ABB RobotStudio station: SmartComponentSolution_20201017-192109.rsstn

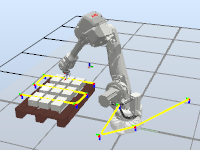
Station SmartComponentSolution (saved by RobotStudio 20.2.9116.0)
Controller IRB_4600_60kg_2.05m, task T_ROB1: task frame (RAPID world) sits at (1429.89, 1152.71, -186.83) mm in the station
Controller IRB_4600_60kg_2.05m
  mechanical unit ROB_1: IRB4600_60_205_C_01, 6 joints, base frame (0, 0, 0) mm
Layout (positions relative to the parent item):
  - IRB4600_60_205_C_01 [mechanism, from Robots\IRB4600_60_205_C_G_01.rslib] at (1429.89, 1152.71, -186.83) mm; joint values [-1.8714, 0.3114, 0.6168, 0, 0.6426, 1.2702] (rad or m)
  - SC_VacuumGripper [smart component] at (3099.75, 399.59, 421.5) mm, rotated rx -180 ry 0 rz 0 deg
      signals: DI diAttach, DO doAttached
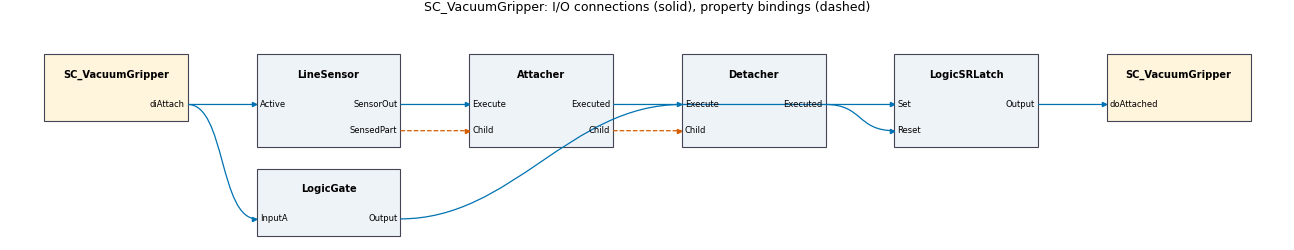
      connections:
        SC_VacuumGripper.diAttach -> LineSensor.Active
        LineSensor.SensorOut -> Attacher.Execute
        SC_VacuumGripper.diAttach -> LogicGate.InputA
        LogicGate.Output -> Detacher.Execute
        Attacher.Executed -> LogicSRLatch.Set
        Detacher.Executed -> LogicSRLatch.Reset
        LogicSRLatch.Output -> SC_VacuumGripper.doAttached
        LineSensor.SensedPart => Attacher.Child
        Attacher.Child => Detacher.Child
    - small_suction_gripper_2 [mechanism] at (0, 0, 0.06) mm
        TCP small_suction_gripper at (-62.96, -41.92, 61.7) mm, rotated rx 90 ry 0 rz 0 deg
        links: suction gripper-2_3
    - LineSensor [smart component, from Components\LineSensor.rslib] at (-638.5, 408.61, -364.87) mm
        properties: Start=[0.641250538776752 -0.457606 0.455378]; End=[0.641250538776752 -0.457606 1.042378]; Radius=0.001; SensedPart=(none); SensedPoint=[0 0 0]
      - _sensorPart_ [part]
    - Attacher [smart component, from Components\Attacher.rslib] at (-2215.65, 408.61, -364.87) mm
        properties: Parent=small_suction_gripper_2; Flange=0; Child=(none); Mount=false; Offset=[0 0 0]; Orientation=[0 0 0]
    - Detacher [smart component, from Components\Detacher.rslib] at (-2215.65, 408.61, -364.87) mm
        properties: Child=(none); KeepPosition=true
    - LogicGate [smart component, from Components\LogicGate.rslib] at (-2215.65, 408.61, -364.87) mm
        properties: Operator=NOT; Delay=0
    - LogicSRLatch [smart component, from Components\LogicSRLatch.rslib] at (-2215.65, 408.61, -364.87) mm
  - Connector [part] at (3092.09, 409.19, 399) mm, rotated rx -90 ry 0 rz 0 deg
  - OD1-B100H50I14-S098974 [part] at (3034.65, 447.69, 354.99) mm, rotated rx 0 ry -90 rz -90 deg
  - Box [part] at (1100.5, 246.78, 144.74) mm, rotated rx 90 ry 0 rz 0 deg
  - Euro Pallet [graphiccomponentgroup, from Equipment\Euro Pallet.rslib] at (680.82, -151.09, 0) mm
    - Body 1 [part, from Equipment\Euro Pallet.rslib] at (188.03, -194.52, 0) mm
  - SC_VaccumGripperDetector [smart component, from Libraries\SC_VaccumGripperDetector.rslib] at (1084.56, 38.85, 366.19) mm, rotated rx 180 ry 0 rz 0 deg
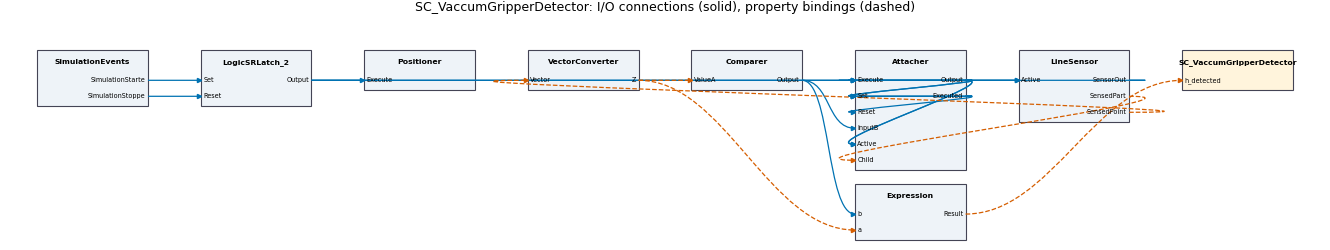
      connections:
        LineSensor.SensorOut -> Attacher.Execute
        LogicGate.Output -> Detacher.Execute
        Attacher.Executed -> LogicSRLatch.Set
        Detacher.Executed -> LogicSRLatch.Reset
        Comparer.Output -> LogicGate_2.InputB
        Comparer.Output -> Expression.b
        LogicGate_3.Output -> LineSensor.Active
        LogicGate_3.Output -> PoseMover.Execute
        SimulationEvents.SimulationStarted -> LogicSRLatch_2.Set
        SimulationEvents.SimulationStopped -> LogicSRLatch_2.Reset
        LogicSRLatch_2.Output -> LineSensor.Active
        LogicSRLatch_2.Output -> PoseMover.Execute
        PoseMover.Executed -> LogicSRLatch_3.Set
        LogicSRLatch_3.Output -> Timer.Active
        Timer.Output -> LogicSRLatch_4.Set
        PoseMover.Executed -> LogicSRLatch_4.Set
        LogicSRLatch_4.Output -> Timer_2.Active
        Timer_2.Output -> LogicSRLatch_5.Set
        LogicSRLatch_5.Output -> PoseMover_2.Execute
        LogicSRLatch_2.Output -> Positioner.Execute
        LineSensor.SensedPart => Attacher.Child
        LineSensor.SensedPoint => VectorConverter.Vector
        VectorConverter.Z => Comparer.ValueA
        VectorConverter.Z => Expression.a
        Expression.Result => SC_VaccumGripperDetector.h_detected
    - small_suction_gripper_2 [mechanism, from Libraries\SC_VaccumGripperDetector.rslib] at (0, 0, 0.06) mm
    - LineSensor [smart component, from Components\LineSensor.rslib] at (-638.5, 408.61, -364.87) mm
        properties: Start=[0.641250538776752 -0.457606 0.455378]; End=[0.641250538776752 -0.457606 1.042378]; Radius=0.001; SensedPart=Box_2; SensedPoint=[1.08731225585938 0.12761491394043 0.244977081298828]
      - _sensorPart_ [part, from Libraries\SC_VaccumGripperDetector.rslib]
    - Comparer [smart component, from Components\Comparer.rslib]
        properties: ValueA=0.244977081298828; Operator=>; ValueB=0.2
    - VectorConverter [smart component, from Components\VectorConverter.rslib]
        properties: X=1.08731225585938; Y=0.12761491394043; Z=0.244977081298828; Vector=[1.08731225585938 0.12761491394043 0.244977081298828]
    - Expression [smart component, from Components\Expression.rslib]
        properties: Expression=a * b; Result=0.244977081298828; a=0.244977081298828; b=1
    - RapidVariable [smart component, from Components\RapidVariable.rslib]
        properties: DataType=pose; Controller=(none); Task=; Module=; Variable=; Value=0; Position=[0 0 0]; Orientation=[0 0 0]
    - SimulationEvents [smart component, from Components\SimulationEvents.rslib]
    - LogicSRLatch_2 [smart component, from Components\LogicSRLatch.rslib]
    - Positioner [smart component, from Components\Positioner.rslib]
        properties: Object=(none); Position=[0 0 0]; Orientation=[0 0 0]; Reference=Global; ReferenceObject=(none)
  - OD1-B100H50I14-S098974_2 [part] at (1019.45, 86.95, 299.69) mm, rotated rx 0 ry -90 rz -90 deg
  - Connector_2 [part] at (1076.9, 48.45, 343.69) mm, rotated rx -90 ry 0 rz 0 deg
  - Box_2 [part] at (1100.5, 65.48, 144.74) mm, rotated rx 90 ry 0 rz 0 deg
  - Box_3 [part] at (1100.5, -122.34, 144.74) mm, rotated rx 90 ry 0 rz 0 deg
  - Box_4 [part] at (1445.39, 246.78, 144.74) mm, rotated rx 90 ry 0 rz 0 deg
  - Box_5 [part] at (1444.74, 62.09, 144.74) mm, rotated rx 90 ry 0 rz 0 deg
  - Box_6 [part] at (1450.77, -121.77, 144.74) mm, rotated rx 90 ry 0 rz 0 deg
  - Box_7 [part] at (1788.47, 246.78, 144.74) mm, rotated rx 90 ry 0 rz 0 deg
  - Box_8 [part] at (1789.72, 54.43, 144.74) mm, rotated rx 90 ry 0 rz 0 deg
  - Box_9 [part] at (1780.97, -127.61, 144.74) mm, rotated rx 90 ry 0 rz 0 deg
  - Frame_1 [frame] at (5315.41, 808.19, -62.39) mm, rotated rx -180 ry 0 rz 0 deg
Attachment: Connector is attached to DEFAULT-34
Attachment: Frame_1 is attached to SC_VacuumGripper
Attachment: OD1-B100H50I14-S098974 is attached to DEFAULT-34
Attachment: OD1-B100H50I14-S098974_2 is attached to DEFAULT-34
Attachment: Connector_2 is attached to DEFAULT-34
Attachment: SC_VaccumGripperDetector is attached to IRB4600_60_205_C_01 / Link6
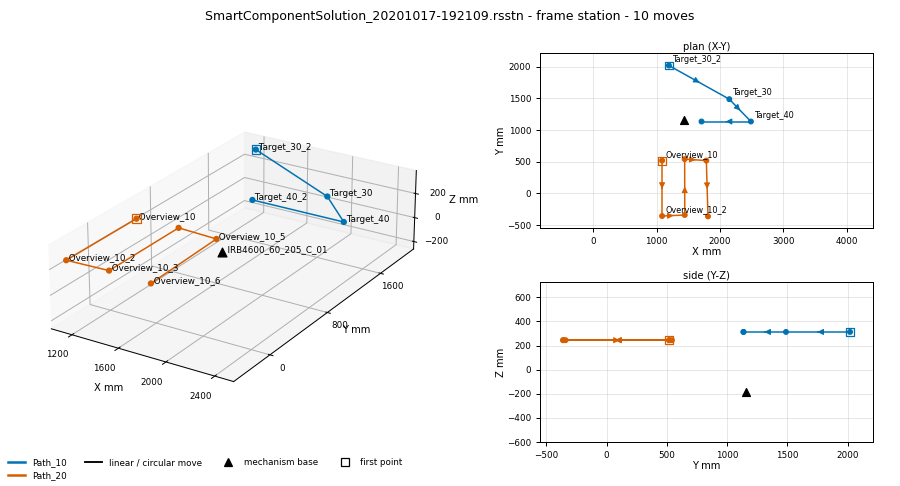
[picture p0: tool path of SmartComponentSolution_20201017-192109.rsstn in frame station, 10 of 10 moves have a stored position in this frame; points joined in program order, loops and branches not executed]
Targets, tools, work objects and paths stored in the station, written as RAPID:
! task T_ROB1
MODULE Module1
  CONST robtarget Target_30:=[[716.121686162,335.077687596,500],[0,1,0,0],[0,0,-2,0],[9E+09,9E+09,9E+09,9E+09,9E+09,9E+09]];
  CONST robtarget Target_40:=[[1057.065915871,-17.60100368,500],[0,1,0,0],[0,-1,-2,0],[9E+09,9E+09,9E+09,9E+09,9E+09,9E+09]];
  CONST robtarget Target_30_2:=[[-237.219768702,866.283675835,500],[0,1,0,0],[0,0,-2,0],[9E+09,9E+09,9E+09,9E+09,9E+09,9E+09]];
  CONST robtarget Target_40_2:=[[277.117965124,-17.60100368,500],[0,1,0,0],[0,0,-2,0],[9E+09,9E+09,9E+09,9E+09,9E+09,9E+09]];
  CONST robtarget Overview_10:=[[-345.337592383,-634.2218361,431.52658222],[0,1,0,0],[0,0,0,0],[9E+09,9E+09,9E+09,9E+09,9E+09,9E+09]];
  CONST robtarget Overview_10_2:=[[-345.337592383,-1509.837410954,431.52658222],[0,1,0,0],[0,0,0,0],[9E+09,9E+09,9E+09,9E+09,9E+09,9E+09]];
  CONST robtarget Overview_10_3:=[[12.284555899,-1493.428131522,431.52658222],[0,1,0,0],[0,0,0,0],[9E+09,9E+09,9E+09,9E+09,9E+09,9E+09]];
  CONST robtarget Overview_10_4:=[[11.425088297,-611.443739064,431.52658222],[0,1,0,0],[0,0,0,0],[9E+09,9E+09,9E+09,9E+09,9E+09,9E+09]];
  CONST robtarget Overview_10_5:=[[353.203433771,-634.2218361,431.52658222],[0,1,0,0],[0,0,0,0],[9E+09,9E+09,9E+09,9E+09,9E+09,9E+09]];
  CONST robtarget Overview_10_6:=[[379.156403723,-1514.983024916,431.52658222],[0,1,0,0],[0,0,0,0],[9E+09,9E+09,9E+09,9E+09,9E+09,9E+09]];
  PROC Path_10()
    MoveL Target_30_2,v1000,z100,small_suction_gripper\WObj:=wobj0;
    MoveL Target_30,v1000,z100,small_suction_gripper\WObj:=wobj0;
    MoveL Target_40,v1000,z100,small_suction_gripper\WObj:=wobj0;
    MoveL Target_40_2,v1000,z100,small_suction_gripper\WObj:=wobj0;
  ENDPROC
  PROC main()
    Path_20;
  ENDPROC
  PROC Path_20()
    MoveL Overview_10,v80,z100,small_suction_gripper\WObj:=wobj0;
    MoveL Overview_10_2,v80,z100,small_suction_gripper\WObj:=wobj0;
    MoveL Overview_10_3,v80,z100,small_suction_gripper\WObj:=wobj0;
    MoveL Overview_10_4,v80,z100,small_suction_gripper\WObj:=wobj0;
    MoveL Overview_10_5,v80,z100,small_suction_gripper\WObj:=wobj0;
    MoveL Overview_10_6,v80,z100,small_suction_gripper\WObj:=wobj0;
  ENDPROC
ENDMODULE

! task T_ROB1
MODULE CalibData
  PERS tooldata small_suction_gripper:=[TRUE,[[-0.000055309,0.000726868,121.499905969],[1,0.000000005,0.000000013,-0.000000029]],[1,[0.443001337,-9.457000743,69.908999891],[1,0,0,0],0,0,0]];
ENDMODULE

